// TIA Portal V17 export
// export: Created 2022-07-28T18:03:17.838381Z, ExportSetting None, DisplayName Totally Integrated Automation Portal, DisplayVersion V17, DisplayName TIA Portal Openness, DisplayVersion V17, DisplayName TIA Portal Teamcenter Gateway, DisplayVersion V17, DisplayName TIA Portal Version Control Interface, DisplayVersion V17, DisplayName TIA Portal Test Suite Advanced, DisplayVersion V17, DisplayName SINAMICS Startdrive Advanced, DisplayVersion V17, DisplayName SINAMICS DCC, DisplayVersion V17, DisplayName SINAMICS Startdrive G130, G150, S120, S150, SINAMICS MV, S210, DisplayVersion V17, DisplayName SINAMICS Startdrive G110M, G120, G120C, G120D, G120P, G115D, DisplayVersion V17, DisplayName STEP 7 Professional, DisplayVersion V17, DisplayName SIMATIC Energy Suite, DisplayVersion V17, DisplayName STEP 7 CFC, DisplayVersion V17, DisplayName STEP 7 Safety, DisplayVersion V17, DisplayName WinCC Advanced / Unified PC, DisplayVersion V17, DisplayName SIMATIC Visualization Architect, DisplayVersion V17
TYPE "_AutoControl_ElementSTW"
   STRUCT
      Fault : Bool;   // 1 = Fault is present
      Ready : Bool;   // 1 = Element ready for start
      ControlAchieve : Bool;   // 1 = Set control command is achieved
      InOtherRoutAvailable : Bool;   // 1 = Element using in some routs, but available for use in other
      InOtherRoutUnavailable : Bool;   // 1 = Element using in some routs, but not available for use in other
      StartPID : Bool;
      StartFull : Bool;
      bit7 : Bool;
      bit8 : Bool;
      bit9 : Bool;
      bit10 : Bool;
      bit11 : Bool;
      bit12 : Bool;
      bit13 : Bool;
      bit14 : Bool;
      bit15 : Bool;
      Release : Bool;   // 1 = Release for start element in auto mode. Set in auto block, reset in element block (life bit)
      bit17 : Bool := FALSE;
      bit18 : Bool := FALSE;
      bit19 : Bool := FALSE;
      bit20 : Bool := FALSE;
      bit21 : Bool := FALSE;
      bit22 : Bool := FALSE;
      bit23 : Bool := FALSE;
      bit24 : Bool := FALSE;
      bit25 : Bool := FALSE;
      bit26 : Bool := FALSE;
      bit27 : Bool := FALSE;
      bit28 : Bool := FALSE;
      bit29 : Bool := FALSE;
      bit30 : Bool := FALSE;
      bit31 : Bool := FALSE;
   END_STRUCT;
END_TYPE
